TEXTLIST TL_E_INSTANCE_CMD
  0 = 'NULL'
  1 = 'INIT'
  2 = 'DISABLE'
  3 = 'ENABLE'
  4 = 'WORK'
  102 = 'CLEAR'
   = ''
END_TEXTLIST

(* stored: Version 1.1.0.1
   TextList TL_E_INSTANCE_CMD: Id {d6ba9340-1698-4061-aab9-10da4232e43a} *)
